// TIA Portal project "PartidaEstrelaTrianguloReversao" (V17)

(* hardware
DEVICE "S7-1200 station_1"  S7-1200 Station
   slot 0: "Rack_0"  S7-1200 Rack  Rack  V1.0
   slot 1: "PLC_EstrelaTriangulo"  CPU 1214C DC/DC/DC  6ES7 214-1AG40-0XB0  V4.2
   slot 3: "AQ 1x12BIT_1"  AQ1 signal board  6ES7 232-4HA30-0XB0  V1.0
   slot 101: "CM 1241 (RS485)_1"  CM 1241 (RS485)  6ES7 241-1CH30-0XB0  V1.0
*)

// ===== PLC "PLC_EstrelaTriangulo"  CPU 1214C DC/DC/DC =====

VAR_GLOBAL   // PLC tag table "Default tag table"
   "K2" AT %Q0.1 : Bool;
   "Desliga" AT %I0.1 : Bool;
   "Seletora" AT %I0.0 : Bool;
   "Liga" AT %I0.2 : Bool;
   "K1" AT %Q0.0 : Bool;
   "Tag_1" AT %I0.5 : Bool;
   "K3" AT %Q0.2 : Bool;
   "K4" AT %Q0.3 : Bool;
   "MK4" AT %M0.0 : Bool;
   "MK4.1" AT %M0.1 : Bool;
   "MK3" AT %M0.2 : Bool;
   "MK3.1" AT %M0.3 : Bool;
END_VAR

// folder: System blocks/Program resources

DATA_BLOCK "Contador_1"   // DB1
{ S7_Optimized_Access := 'TRUE' }
AUTHOR : Simatic
FAMILY : IEC
NAME : CNTR
VERSION : 1.0
// stored: InstanceOfName IEC_COUNTER
"IEC_COUNTER"
BEGIN
END_DATA_BLOCK

DATA_BLOCK "Timer_1"   // DB2
{ S7_Optimized_Access := 'TRUE' }
AUTHOR : Simatic
FAMILY : IEC
NAME : IEC_TMR
VERSION : 1.0
// stored: InstanceOfName IEC_TIMER
"IEC_TIMER"
BEGIN
END_DATA_BLOCK

DATA_BLOCK "Timer_2"   // DB3
{ S7_Optimized_Access := 'TRUE' }
AUTHOR : Simatic
FAMILY : IEC
NAME : IEC_TMR
VERSION : 1.0
// stored: InstanceOfName IEC_TIMER
"IEC_TIMER"
BEGIN
END_DATA_BLOCK

DATA_BLOCK "Timer_Delay_k3"   // DB4
{ S7_Optimized_Access := 'TRUE' }
AUTHOR : Simatic
FAMILY : IEC
NAME : IEC_TMR
VERSION : 1.0
// stored: InstanceOfName IEC_TIMER
"IEC_TIMER"
BEGIN
END_DATA_BLOCK

DATA_BLOCK "IEC_Timer_1"   // DB5
{ S7_Optimized_Access := 'TRUE' }
AUTHOR : Simatic
FAMILY : IEC
NAME : IEC_TMR
VERSION : 1.0
// stored: InstanceOfName IEC_TIMER
"IEC_TIMER"
BEGIN
END_DATA_BLOCK

// folder: (top level)

ORGANIZATION_BLOCK "Main"   // OB1, LAD, ProgramCycle
TITLE = "Main Program Sweep (Cycle)"
{ S7_Optimized_Access := 'TRUE' }
VERSION : 0.1
// Partida estrela triangulo com reversão
   VAR_INPUT
      Initial_Call : Bool;   // Initial call of this OB
      Remanence : Bool;   // =True, if remanent data are available
   END_VAR
BEGIN

REGION Network 1: Liga K1
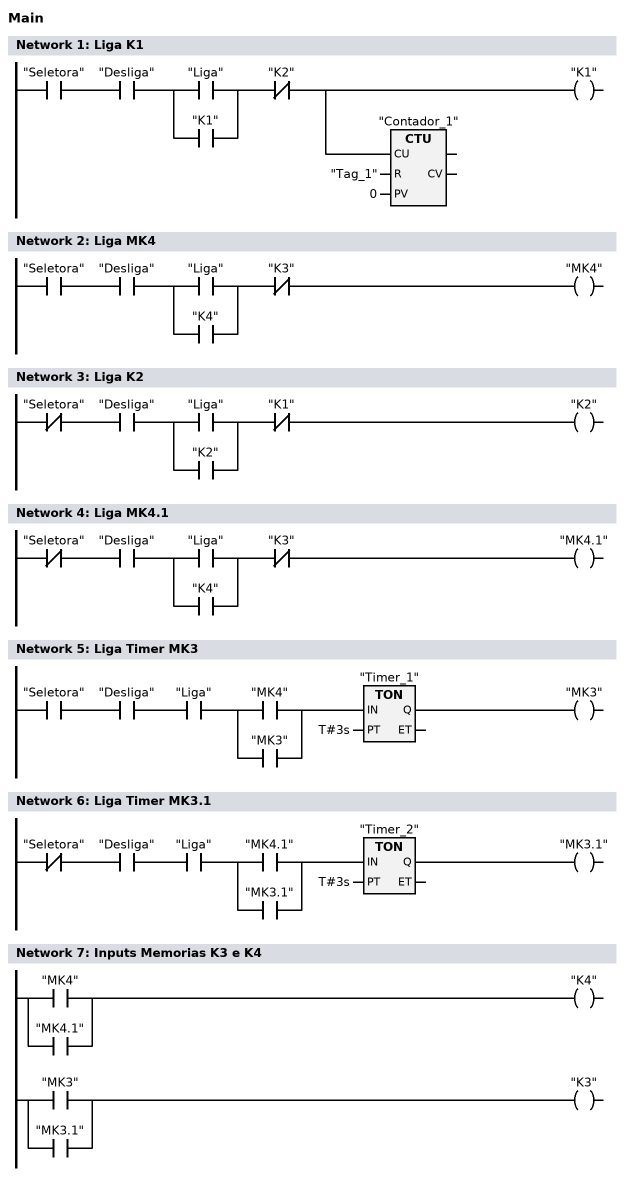
   "K1" := "Seletora" AND "Desliga" AND ("Liga" OR "K1") AND NOT "K2";
   "Contador_1".CTU(CU := "K1", R := "Tag_1", PV := 0);
END_REGION

REGION Network 2: Liga MK4
   RUNG wire#powerrail
      Contact( "Seletora" )
      Contact( "Desliga" )
      wire#w1
      Contact( "Liga" )
      wire#w2
      I_Contact( "K3" )
      Coil( "MK4" )
   END_RUNG
   RUNG wire#w1
      Contact( "K4" )
   END_RUNG wire#w2
   // the same network as SCL:
   "MK4" := "Seletora" AND "Desliga" AND ("Liga" OR "K4") AND NOT "K3";
END_REGION

REGION Network 3: Liga K2
   RUNG wire#powerrail
      I_Contact( "Seletora" )
      Contact( "Desliga" )
      wire#w1
      Contact( "Liga" )
      wire#w2
      I_Contact( "K1" )
      Coil( "K2" )
   END_RUNG
   RUNG wire#w1
      Contact( "K2" )
   END_RUNG wire#w2
   // the same network as SCL:
   "K2" := NOT "Seletora" AND "Desliga" AND ("Liga" OR "K2") AND NOT "K1";
END_REGION

REGION Network 4: Liga MK4.1
   RUNG wire#powerrail
      I_Contact( "Seletora" )
      Contact( "Desliga" )
      wire#w1
      Contact( "Liga" )
      wire#w2
      I_Contact( "K3" )
      Coil( "MK4.1" )
   END_RUNG
   RUNG wire#w1
      Contact( "K4" )
   END_RUNG wire#w2
   // the same network as SCL:
   "MK4.1" := NOT "Seletora" AND "Desliga" AND ("Liga" OR "K4") AND NOT "K3";
END_REGION

REGION Network 5: Liga Timer MK3
   "Timer_1".TON(IN := "Seletora" AND "Desliga" AND "Liga" AND ("MK4" OR "MK3"), PT := T#3s);
   "MK3" := "Timer_1".Q;
END_REGION

REGION Network 6: Liga Timer MK3.1
   "Timer_2".TON(IN := NOT "Seletora" AND "Desliga" AND "Liga" AND ("MK4.1" OR "MK3.1"), PT := T#3s);
   "MK3.1" := "Timer_2".Q;
END_REGION

REGION Network 7: Inputs Memorias K3 e K4
   RUNG wire#powerrail
      Contact( "MK4" )
      wire#w1
      Coil( "K4" )
   END_RUNG
   RUNG wire#powerrail
      Contact( "MK4.1" )
   END_RUNG wire#w1
   RUNG wire#powerrail
      Contact( "MK3" )
      wire#w2
      Coil( "K3" )
   END_RUNG
   RUNG wire#powerrail
      Contact( "MK3.1" )
   END_RUNG wire#w2
   // the same network as SCL:
   "K4" := "MK4" OR "MK4.1";
   "K3" := "MK3" OR "MK3.1";
END_REGION
END_ORGANIZATION_BLOCK

ORGANIZATION_BLOCK "Main_1"   // OB123, SCL, ProgramCycle
TITLE = "Main Program Sweep (Cycle)"
{ S7_Optimized_Access := 'TRUE' }
VERSION : 0.1
   VAR_INPUT
      Initial_Call : Bool;   // Initial call of this OB
      Remanence : Bool;   // =True, if remanent data are available
   END_VAR
BEGIN
   IF "Seletora" = TRUE AND "Desliga" = TRUE AND "Liga" = TRUE THEN
       // Statement section IF
       "K1" := TRUE;
       "K4" := TRUE;
   ELSIF "Seletora" = FALSE THEN
       "K1" := FALSE;
       "K4" := FALSE;
   ELSIF "Desliga" = FALSE THEN
       "K1" := FALSE;
       "K4" := FALSE;
   END_IF;

   "IEC_Timer_1".TON(IN:="K4",
                     PT:=T#5s,
                     Q=>"K3");

   IF "K3" = TRUE THEN
       "K4" := FALSE;
   END_IF;
END_ORGANIZATION_BLOCK